FUNCTION_BLOCK Machine EXTENDS FB_PackML_BaseModule
VAR
	CamModule : CamModule := (Name := 'Cam Module');
END_VAR

// Automatically enables and disables HMI control based on the PackML mode
METHOD PROTECTED HMIPermissions

// This method is called cyclically by CyclicLogic()
AllowHMIControl(TRUE);
END_METHOD

// Basic module initialization logic
METHOD PROTECTED Initialize : BOOL;

// This method is called by CyclicLogic() as required
Initialize := FALSE;
CASE DescendantSequenceState OF
	0:
		RegisterSubmodule(SubModule := CamModule);
		DescendantSequenceState := DescendantSequenceState + 10;

	10:
		IF SUPER^.Initialize() THEN
			Initialize := TRUE;
		END_IF
END_CASE
END_METHOD

END_FUNCTION_BLOCK

(* stored: Version 1.1.0.1, ProductVersion 3.1.4024.12
   POU Machine: Id {f0bb7911-80d1-477d-8de7-ffb3a7f394bb}, SpecialFunc None
   Method HMIPermissions: Id {a511af05-b33e-4341-90d7-f7134d2e90db}
   Method Initialize: Id {009da281-27b7-48c7-b1db-982fe18ad8aa} *)
